DATA_BLOCK "DbFlowControl"	// DB 231
TITLE = 'Значения параметров БУ ВН2012'
AUTHOR : Konst
FAMILY : Main
NAME : DbCalc
VERSION : 0.0
  STRUCT
   Calc_NumHour : INT ;	//номер расчетного часа в сутках ([[1-24])
   Calc_NumDay : INT ;	//номер расчетного дня в месяце ([[1-31])
   BoundBuCount : REAL ;	//Граница X зацикленного счётчика РГ за сезон в БУ : [1-X]
   HmiNum_To_Copy : INT ;	//какой элемент из DbFlowData копировать в 0-й (0-скопировано\[1-7]-запрос)
   Num_In_Copy : INT ;	//номер скопированного эл-та
   TimeStamp_Copy : DATE_AND_TIME ;	//метка времени в момент копирования
   Ev_Hour_Next : BOOL ;	//#событие : наступление нового часа
   Ev_Day_Next : BOOL ;	//#событие : наступление новых расчетных суток
   Ev_Month_Next : BOOL ;	//#событие : наступление нового расчетного месяца
   lblCalc_Hour_Prev : BOOL ;	//обновление расчёта за предыд. час: 1-момент наступил\0-нет
   lblCalc_Day_Prev : BOOL ;	//обновление счётчика за предыд. день: 1-момент наступил\0-нет
   lblCalc_Month_Prev : BOOL ;	//обновление счётчика за предыд. месяц: 1-момент наступил\0-нет
   Reset_Data_All : BOOL ;	//+инициализация данных по всем эл-там FlowData[] : 1-да \0-нет
   NonStop_Copy : BOOL ;	//+безостановочное копирование в 0-й эл-т: 1-non-stop\0- 1 раз
   NumHour : INT ;	//+количество элементов в Flow_Hour_Arc[]
   NumDay : INT ;	//+количество элементов в Flow_Day_Arc[]
   NumMonth : INT ;	//+количество элементов в Flow_Month_Arc[]
   Num_Hour_Current : INT ;	//+номер текущего часа с момента EventH
   Num_Hour_Prev : INT ;	//+номер предыдущего часа с момента EventH (или LastWork)
   Num_Day_Current : INT ;	//+номер i текущих расчетных суток для Flow_Day_Arc[i]
   Num_Day_Prev : INT ;	//+номер i новых расчетных суток для Flow_Day_Arc[i]
   Num_Month_Current : INT ;	//+номер i текущего расчетного месяца для Flow_Month_Arc[i]
   Num_Month_Prev : INT ;	//+номер i нового расчетного месяца для Flow_Month_Arc[i]
  END_STRUCT ;	//Db
BEGIN
   Calc_NumHour := 10;
   Calc_NumDay := 1;
   BoundBuCount := 9.000000e+05;
   NumHour := 48;
   NumDay := 31;
   NumMonth := 12;
END_DATA_BLOCK

DATA_BLOCK "DbSepBlow"	// DB 232
VERSION : 0.0
  STRUCT
   numSep : INT ;	// количество сепараторов
   BlowCountMax : INT ;
   dzTimeScan : INT ;	//время сканирования данных по РЖ в МСек
   SepBlowParam : ARRAY  [1 .. 3 ] OF UDT 211;
  END_STRUCT ;	//Db
BEGIN
   numSep := 3;
   BlowCountMax := 5000;
   dzTimeScan := 1000;
   SepBlowParam[1].ControlObject := 1;
   SepBlowParam[1].WaterLevel_LoControl := 3.750000e+01;
   SepBlowParam[1].WaterLevel_HiControl := 5.000000e+01;
   SepBlowParam[1].BlowTimeDurationMax := 120;
   SepBlowParam[1].BlowTimeIntervalMax := 1000;
   SepBlowParam[1].BlowTypeAuto := TRUE;
   SepBlowParam[1].Flow_Sens_Correct_Cut := 5.000000e-02;
   SepBlowParam[1].Flow_Sens_Correct_0 := 3.000000e-02;
   SepBlowParam[1].Tm_Valve_FullClose := 30;
   SepBlowParam[2].ControlObject := 1;
   SepBlowParam[2].WaterLevel_LoControl := 3.750000e+01;
   SepBlowParam[2].WaterLevel_HiControl := 5.000000e+01;
   SepBlowParam[2].BlowTimeDurationMax := 120;
   SepBlowParam[2].BlowTimeIntervalMax := 1000;
   SepBlowParam[2].BlowTypeAuto := TRUE;
   SepBlowParam[2].Flow_Sens_Correct_Cut := 5.000000e-02;
   SepBlowParam[2].Flow_Sens_Correct_0 := 3.000000e-02;
   SepBlowParam[2].Tm_Valve_FullClose := 30;
   SepBlowParam[3].ControlObject := 1;
   SepBlowParam[3].WaterLevel_LoControl := 3.750000e+01;
   SepBlowParam[3].WaterLevel_HiControl := 5.000000e+01;
   SepBlowParam[3].BlowTimeDurationMax := 120;
   SepBlowParam[3].BlowTimeIntervalMax := 1000;
   SepBlowParam[3].BlowTypeAuto := TRUE;
   SepBlowParam[3].Flow_Sens_Correct_Cut := 5.000000e-02;
   SepBlowParam[3].Flow_Sens_Correct_0 := 3.000000e-02;
   SepBlowParam[3].Tm_Valve_FullClose := 30;
END_DATA_BLOCK

DATA_BLOCK "DbCaution"	// DB 233
VERSION : 0.0
  STRUCT
   numCaution : INT ;	// количество тревог, описанных в CautionParam[]
   ValueID : INT ;	//значение ID последней (предыдущей) тревоги
   isActive : BOOL ;	// метка активности (необх-ти проигрывания) последней тревоги: 0-нет\1- активна
   MelodyBuffer : WORD ;	// переменная для "проигрывания" тревоги
   SignalW : BOOL ;	// значение DO-сигнала для упр. светом и звуком: 0-выкл\ 1- включить
   tStamp_Format_TOD : TIME_OF_DAY ;	//метка времени в момент возникн. последней тревоги в формате TOD
   tStamp_Format_Str : STRING  [17 ];	//метка времени в строковом формате "DD.MM.YY HH:MM:SS"
   CautionParam : ARRAY  [1 .. 6 ] OF UDT 212;
  END_STRUCT ;	//Db
BEGIN
   numCaution := 6;
   CautionParam[1].Melody := 693;
   CautionParam[1].PlayOn_SepSignal_Zvuk1 := TRUE;
   CautionParam[1].PlayOn_OperSignal_Zvuk := TRUE;
   CautionParam[2].Melody := 693;
   CautionParam[2].PlayOn_SepSignal_Svet1 := TRUE;
   CautionParam[2].PlayOn_SepSignal_Svet2 := TRUE;
   CautionParam[2].PlayOn_SepSignal_Zvuk1 := TRUE;
   CautionParam[2].PlayOn_OperSignal_Svet := TRUE;
   CautionParam[2].PlayOn_OperSignal_Zvuk := TRUE;
   CautionParam[2].PlayOn_UouSignal_Svet := TRUE;
   CautionParam[3].Melody := 693;
   CautionParam[4].Melody := 693;
   CautionParam[4].PlayOn_SepSignal_Svet1 := TRUE;
   CautionParam[4].PlayOn_SepSignal_Svet2 := TRUE;
   CautionParam[4].PlayOn_SepSignal_Zvuk1 := TRUE;
   CautionParam[5].Melody := 693;
   CautionParam[5].PlayOn_OperSignal_Svet := TRUE;
   CautionParam[5].PlayOn_OperSignal_Zvuk := TRUE;
   CautionParam[6].Melody := 693;
   CautionParam[6].PlayOn_UouSignal_Svet := TRUE;
END_DATA_BLOCK

DATA_BLOCK "DbEnum"	// DB 234
VERSION : 0.0
  STRUCT 	//23456789012345678901234
   CAUT_OverMaxTimeBlow : INT ;	// Превышение max длительности продувки

   RBC_AvOst : INT ;	// reasonBanControl : Аварийный останов для всей подсистемы УПС [1-10]
   RBC_RegimRemont : INT ;	// reasonBanControl : режим "Ремонт" для всей подсистемы УПС
  END_STRUCT ;	//Db
BEGIN
   CAUT_OverMaxTimeBlow := 1;
   RBC_AvOst := 1;
   RBC_RegimRemont := 2;
END_DATA_BLOCK

DATA_BLOCK "DbSipValveDeb"	// DB 248
VERSION : 0.0
  STRUCT
   SipValveParam : ARRAY  [1 .. 5 ] OF UDT 248;
  END_STRUCT ;	//Db
BEGIN
END_DATA_BLOCK

DATA_BLOCK "DbKranPpuDeb"	// DB 249
TITLE = 'Значения параметров'
AUTHOR : Konst
FAMILY : Main
NAME : DbKranP2
VERSION : 0.0
  STRUCT
   KranPpuParam : ARRAY  [1 .. 15 ] OF UDT 249;	// м. еще размерность или KranPpuParam_Prev
  END_STRUCT ;	//Db
BEGIN
END_DATA_BLOCK

DATA_BLOCK "idb_fb_ParScan"	// DB 251
AUTHOR : Konst
FAMILY : Main
VERSION : 0.0
"fb_ParScan"
BEGIN
END_DATA_BLOCK

DATA_BLOCK "idb_fb_KranPpu"	// DB 252
AUTHOR : Konst
FAMILY : Main
VERSION : 0.0
"fb_KranPpu"
BEGIN
END_DATA_BLOCK

DATA_BLOCK "idb_fb_Watch"	// DB 253
AUTHOR : Konst
FAMILY : Main
VERSION : 0.0
"fb_Watch"
BEGIN
END_DATA_BLOCK

DATA_BLOCK "idb_fb_ExecCmd"	// DB 254
AUTHOR : Konst
FAMILY : Main
VERSION : 0.0
"fb_ExecCmd"
BEGIN
END_DATA_BLOCK

DATA_BLOCK "idb_fb_SipValve"	// DB 255
AUTHOR : Konst
FAMILY : Main
VERSION : 0.0
"fb_SipValve"
BEGIN
END_DATA_BLOCK

DATA_BLOCK "idb_fb_Flow"	// DB 256
AUTHOR : Konst
FAMILY : Main
VERSION : 0.0
"fb_Flow"
BEGIN
END_DATA_BLOCK

DATA_BLOCK DB 291
AUTHOR : Konst
FAMILY : Main
VERSION : 0.0
FB 291
BEGIN
END_DATA_BLOCK

DATA_BLOCK "db_BSEND"	// DB 292
AUTHOR : SIMATIC
FAMILY : COM_FUNC
VERSION : 0.0
"BSEND"
BEGIN
END_DATA_BLOCK

DATA_BLOCK "db_BRCV"	// DB 293
AUTHOR : SIMATIC
FAMILY : COM_FUNC
VERSION : 0.0
"BRCV"
BEGIN
END_DATA_BLOCK

DATA_BLOCK "DbCpBufSend"	// DB 294
TITLE = 'Области передачи данных'
AUTHOR : Konst
FAMILY : Main
VERSION : 0.0
  STRUCT
   mSendPar : ARRAY  [1 .. 6 ] OF STRUCT
    DevAddr : BYTE ;
    FuncCode : BYTE ;
    DataStartAdr : WORD ;
    DataKol : INT ;
   END_STRUCT ;
  END_STRUCT ;	// Db
BEGIN
   mSendPar[1].DevAddr := B#16#2;
   mSendPar[1].FuncCode := B#16#1;
   mSendPar[1].DataStartAdr := W#16#64;
   mSendPar[1].DataKol := 75;
   mSendPar[2].DevAddr := B#16#2;
   mSendPar[2].FuncCode := B#16#2;
   mSendPar[2].DataStartAdr := W#16#3E8;
   mSendPar[2].DataKol := 240;
   mSendPar[3].DevAddr := B#16#2;
   mSendPar[3].FuncCode := B#16#3;
   mSendPar[3].DataStartAdr := W#16#7D0;
   mSendPar[3].DataKol := 86;
   mSendPar[4].DevAddr := B#16#4;
   mSendPar[4].FuncCode := B#16#1;
   mSendPar[4].DataStartAdr := W#16#6D;
   mSendPar[4].DataKol := 1;
   mSendPar[5].DevAddr := B#16#3D;
   mSendPar[5].FuncCode := B#16#43;
   mSendPar[5].DataStartAdr := W#16#7034;
   mSendPar[5].DataKol := 13361;
   mSendPar[6].DataStartAdr := W#16#2441;
   mSendPar[6].DataKol := 12365;
END_DATA_BLOCK

DATA_BLOCK "DbCpBufRcv"	// DB 295
TITLE = 'Области приема данных'
AUTHOR : Konst
FAMILY : Main
VERSION : 0.0
  STRUCT
   RcvDataFloat : ARRAY  [1 .. 100 ] OF WORD ;
   RcvDataBool : ARRAY  [1 .. 100 ] OF BOOL ;
   RcvDataInt : ARRAY  [1 .. 100 ] OF BYTE ;
  END_STRUCT ;	// Db
BEGIN
END_DATA_BLOCK

ORGANIZATION_BLOCK "obMain"	// OB 1
TITLE = Основной управляющий блок
AUTHOR : Konst
FAMILY : Main
NAME : Main1
VERSION : 1.0
VAR_TEMP
  Info : ARRAY  [0 .. 19 ] OF BYTE ;
  i1 : INT ;
END_VAR
BEGIN
// body was compiled from an SCL source; compiled code not shown
END_ORGANIZATION_BLOCK

ORGANIZATION_BLOCK "obCyclicCalcFlow"	// OB 32
TITLE = Restart CPU
AUTHOR : Konst
FAMILY : Main
NAME : Main1
VERSION : 1.0
VAR_TEMP
  Info : ARRAY  [0 .. 19 ] OF BYTE ;
  i1 : INT ;
  n1 : INT ;
END_VAR
BEGIN
// body was compiled from an SCL source; compiled code not shown
END_ORGANIZATION_BLOCK

ORGANIZATION_BLOCK "obErrRunTime"	// OB 80
TITLE = Restart CPU
AUTHOR : Konst
FAMILY : Main
NAME : Main1
VERSION : 1.0
VAR_TEMP
  Info : ARRAY  [0 .. 19 ] OF BYTE ;
  i1 : INT ;
  n1 : INT ;
END_VAR
BEGIN
// body was compiled from an SCL source; compiled code not shown
END_ORGANIZATION_BLOCK

ORGANIZATION_BLOCK "obRestart"	// OB 100
TITLE = Restart CPU
AUTHOR : Konst
FAMILY : Main
NAME : Main1
VERSION : 1.0
VAR_TEMP
  Info : ARRAY  [0 .. 19 ] OF BYTE ;
  i1 : INT ;
  n1 : INT ;
END_VAR
BEGIN
// body was compiled from an SCL source; compiled code not shown
END_ORGANIZATION_BLOCK
